(* Logix 5000 project; controller Timers Emulate 5570 rev 33.11; software revision 33.00 *)

TASK T00_MainTask (continuous, watchdog 500 ms) : P00_MainProgram

MODULES
   Local : Emulate 5570 (ICP 2, rev 33.11)
END_MODULES

PROGRAM P00_MainProgram   (* main routine R00_MainRoutine *)
VAR
   B01_Activacion_Alarma : BOOL[32];   // BOOL
   ES : BOOL[32];   // Boton de Paro de emergencia
   I01_Desactivar_Alarma : BOOL[32];   // Boton para desactivar Alarma
   I02_Arranque_Centrifugado : BOOL[32];   // Boton de Arranque del Calentador
   I03_Arranque_Lavadora : BOOL[32];
   I99 : BOOL[32];
   O01_Lampara : BOOL[32];   // Luz de seguridad
   O02_Alarma : BOOL[32];   // Alarma
   O03_Centrifugadora : BOOL[32];   // Encendido de Centrifugadora
   O04_Frenos : BOOL[32];   // Activacion de Frenos
   O05_SegurosPuerta : BOOL[32];   // Activacion de Seguros Puerta
   O06_Lavador : BOOL[32];   // Activacion de Lavadora
   REST : BOOL[32];
   RTO : BOOL[32];
   S01_Movimiento : BOOL[32];   // Sensor de Movimiento
   T01_DesactivarLuz : TIMER[32] := ([0].PRE := 10000);   // Timer para desactivar luz en 10s
   T02_Alarma : TIMER[32] := ([0].PRE := 5000);   // Activacion de Alarma
   T03_Centrifugado : TIMER[32] := ([0].PRE := 10000);   // Tiempo de centrifugado
   T04_Tiempo_de_Frenado : TIMER[32] := ([0].PRE := 5000);   // Tiempo de frenado
   T05_Tiempo_Lavado : TIMER[32] := ([0].PRE := 15000);   // Tiempo de Lavado
   T06_Tiempo_Uso : TIMER[32] := ([0].PRE := 60000);
   T99_T : TIMER[32] := ([0].PRE := 6000, [0].ACC := 30035);
END_VAR

ROUTINE R00_MainRoutine   (* ladder *)
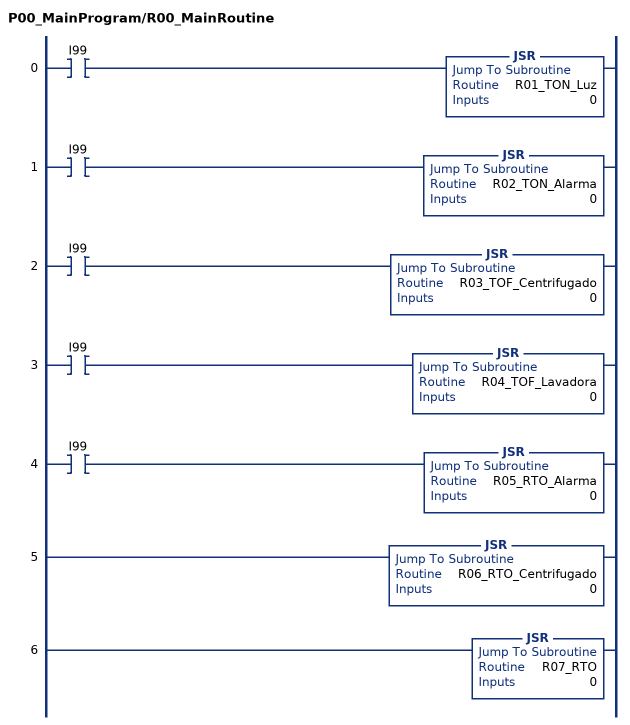
   0: XIC(I99)JSR(R01_TON_Luz,0);
   1: XIC(I99)JSR(R02_TON_Alarma,0);
   2: XIC(I99)JSR(R03_TOF_Centrifugado,0);
   3: XIC(I99)JSR(R04_TOF_Lavadora,0);
   4: XIC(I99)JSR(R05_RTO_Alarma,0);
   5: JSR(R06_RTO_Centrifugado,0);
   6: JSR(R07_RTO,0);
END_ROUTINE

ROUTINE R01_TON_Luz   (* ladder *)
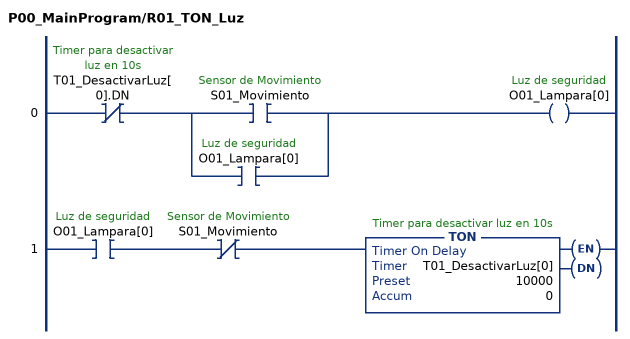
   0: XIO(T01_DesactivarLuz[0].DN)[XIC(S01_Movimiento) ,XIC(O01_Lampara[0]) ]OTE(O01_Lampara[0]);
   1: XIC(O01_Lampara[0])XIO(S01_Movimiento)TON(T01_DesactivarLuz[0],10000,0);
END_ROUTINE

ROUTINE R02_TON_Alarma   (* ladder *)
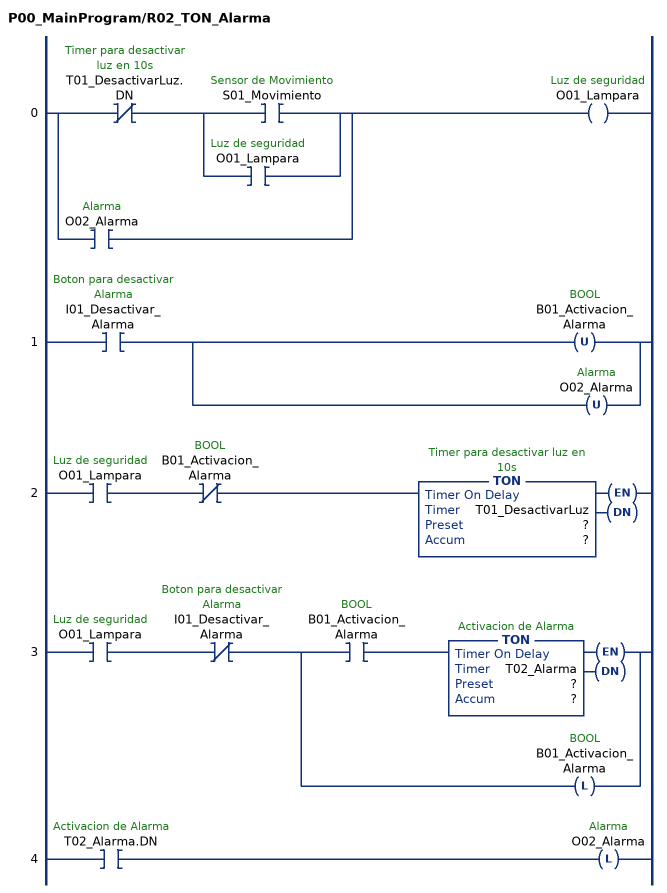
   0: [XIO(T01_DesactivarLuz.DN) [XIC(S01_Movimiento) ,XIC(O01_Lampara) ] ,XIC(O02_Alarma) ]OTE(O01_Lampara);
   1: XIC(I01_Desactivar_Alarma)[OTU(B01_Activacion_Alarma) ,OTU(O02_Alarma) ];
   2: XIC(O01_Lampara)XIO(B01_Activacion_Alarma)TON(T01_DesactivarLuz,?,?);
   3: XIC(O01_Lampara)XIO(I01_Desactivar_Alarma)[XIC(B01_Activacion_Alarma) TON(T02_Alarma,?,?) ,OTL(B01_Activacion_Alarma) ];
   4: XIC(T02_Alarma.DN)OTL(O02_Alarma);
END_ROUTINE

ROUTINE R03_TOF_Centrifugado   (* ladder *)
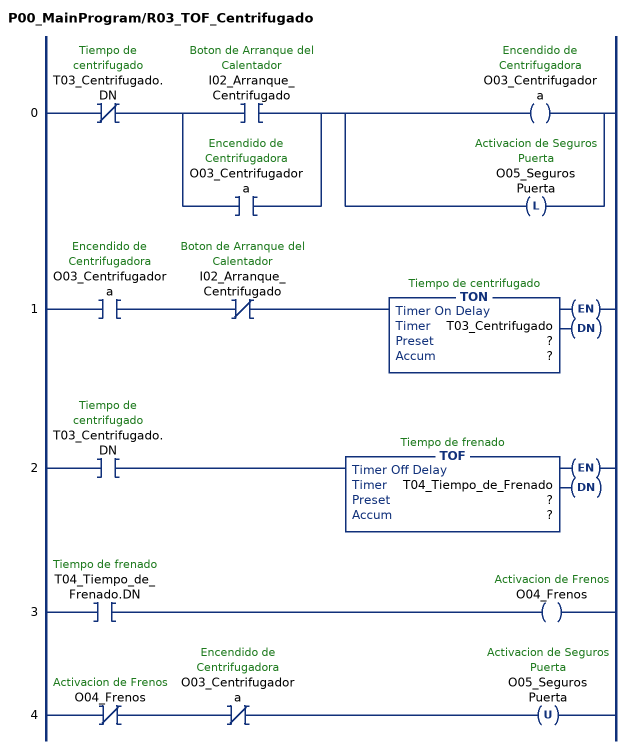
   0: XIO(T03_Centrifugado.DN)[XIC(I02_Arranque_Centrifugado) ,XIC(O03_Centrifugadora) ][OTE(O03_Centrifugadora) ,OTL(O05_SegurosPuerta) ];
   1: XIC(O03_Centrifugadora)XIO(I02_Arranque_Centrifugado)TON(T03_Centrifugado,?,?);
   2: XIC(T03_Centrifugado.DN)TOF(T04_Tiempo_de_Frenado,?,?);
   3: XIC(T04_Tiempo_de_Frenado.DN)OTE(O04_Frenos);
   4: XIO(O04_Frenos)XIO(O03_Centrifugadora)OTU(O05_SegurosPuerta);
END_ROUTINE

ROUTINE R04_TOF_Lavadora   (* ladder *)
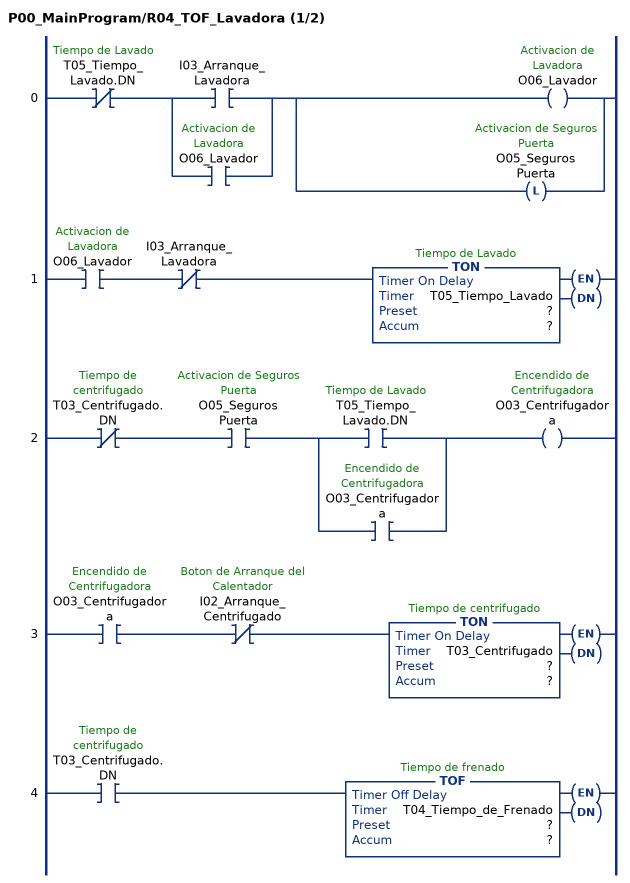
   0: XIO(T05_Tiempo_Lavado.DN)[XIC(I03_Arranque_Lavadora) ,XIC(O06_Lavador) ][OTE(O06_Lavador) ,OTL(O05_SegurosPuerta) ];
   1: XIC(O06_Lavador)XIO(I03_Arranque_Lavadora)TON(T05_Tiempo_Lavado,?,?);
   2: XIO(T03_Centrifugado.DN)XIC(O05_SegurosPuerta)[XIC(T05_Tiempo_Lavado.DN) ,XIC(O03_Centrifugadora) ]OTE(O03_Centrifugadora);
   3: XIC(O03_Centrifugadora)XIO(I02_Arranque_Centrifugado)TON(T03_Centrifugado,?,?);
   4: XIC(T03_Centrifugado.DN)TOF(T04_Tiempo_de_Frenado,?,?);
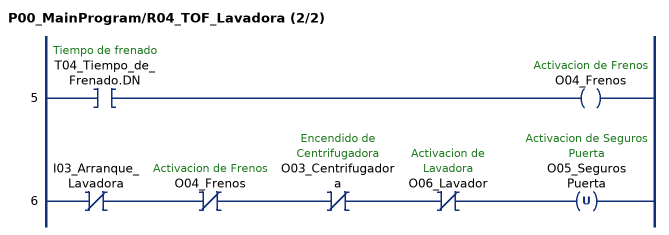
   5: XIC(T04_Tiempo_de_Frenado.DN)OTE(O04_Frenos);
   6: XIO(I03_Arranque_Lavadora)XIO(O04_Frenos)XIO(O03_Centrifugadora)XIO(O06_Lavador)OTU(O05_SegurosPuerta);
END_ROUTINE

ROUTINE R05_RTO_Alarma   (* ladder *)
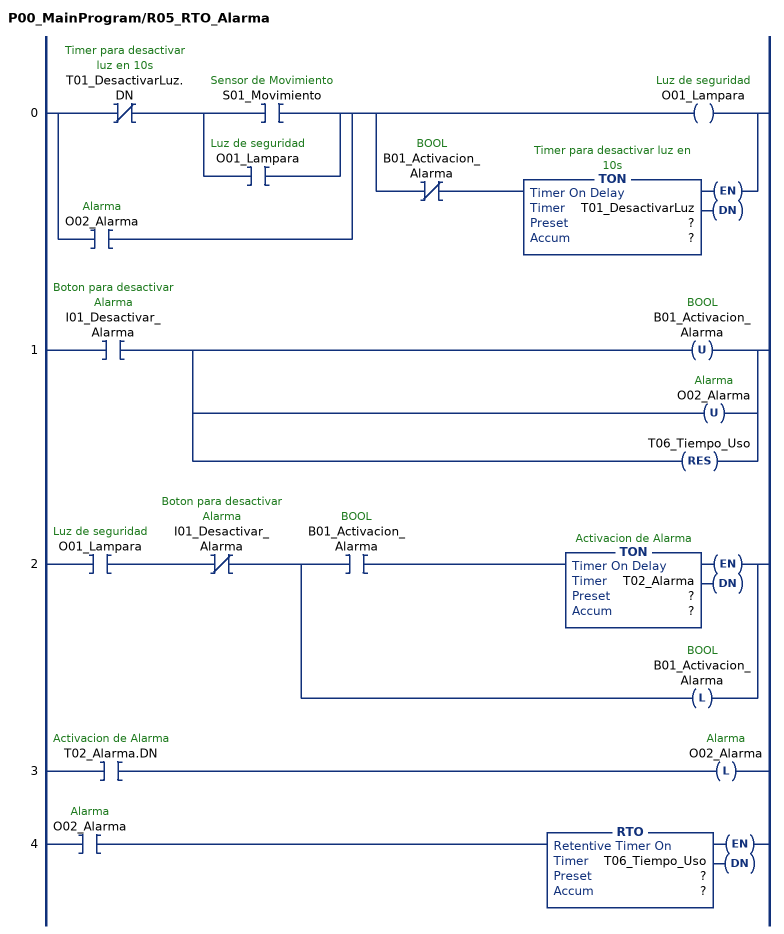
   0: [XIO(T01_DesactivarLuz.DN) [XIC(S01_Movimiento) ,XIC(O01_Lampara) ] ,XIC(O02_Alarma) ][OTE(O01_Lampara) ,XIO(B01_Activacion_Alarma) TON(T01_DesactivarLuz,?,?) ];
   1: XIC(I01_Desactivar_Alarma)[OTU(B01_Activacion_Alarma) ,OTU(O02_Alarma) ,RES(T06_Tiempo_Uso) ];
   2: XIC(O01_Lampara)XIO(I01_Desactivar_Alarma)[XIC(B01_Activacion_Alarma) TON(T02_Alarma,?,?) ,OTL(B01_Activacion_Alarma) ];
   3: XIC(T02_Alarma.DN)OTL(O02_Alarma);
   4: XIC(O02_Alarma)RTO(T06_Tiempo_Uso,?,?);
END_ROUTINE

ROUTINE R06_RTO_Centrifugado   (* ladder *)
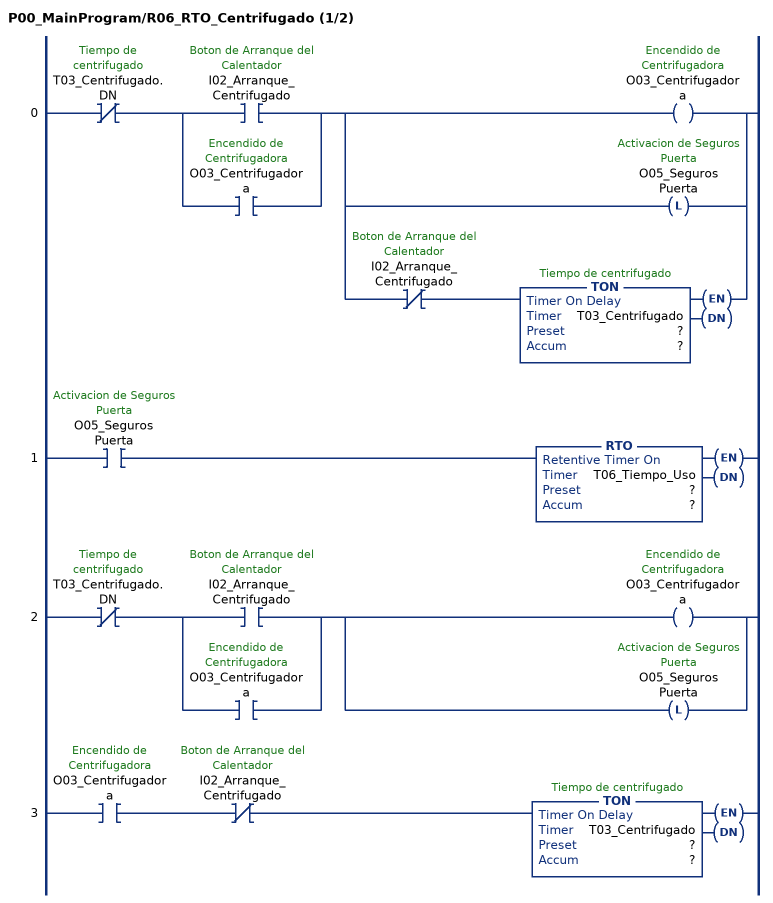
   0: XIO(T03_Centrifugado.DN)[XIC(I02_Arranque_Centrifugado) ,XIC(O03_Centrifugadora) ][OTE(O03_Centrifugadora) ,OTL(O05_SegurosPuerta) ,XIO(I02_Arranque_Centrifugado) TON(T03_Centrifugado,?,?) ];
   1: XIC(O05_SegurosPuerta)RTO(T06_Tiempo_Uso,?,?);
   2: XIO(T03_Centrifugado.DN)[XIC(I02_Arranque_Centrifugado) ,XIC(O03_Centrifugadora) ][OTE(O03_Centrifugadora) ,OTL(O05_SegurosPuerta) ];
   3: XIC(O03_Centrifugadora)XIO(I02_Arranque_Centrifugado)TON(T03_Centrifugado,?,?);
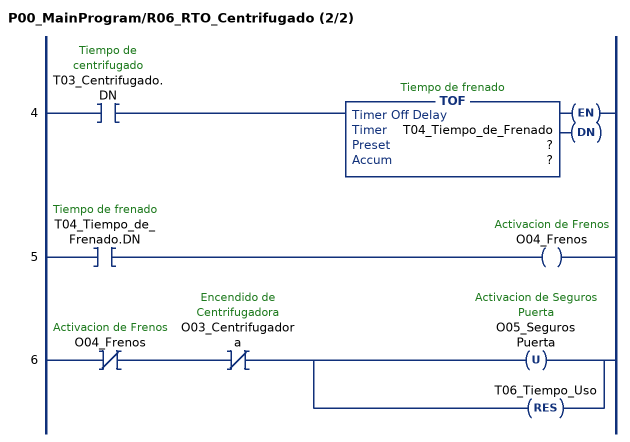
   4: XIC(T03_Centrifugado.DN)TOF(T04_Tiempo_de_Frenado,?,?);
   5: XIC(T04_Tiempo_de_Frenado.DN)OTE(O04_Frenos);
   6: XIO(O04_Frenos)XIO(O03_Centrifugadora)[OTU(O05_SegurosPuerta) ,RES(T06_Tiempo_Uso) ];
END_ROUTINE
END_PROGRAM
